(* CODESYS project TcTransform.library
   DefaultNamespace: TcTransform
   Description: Coordinate system transformation library
   Author: Andrew Burks
   DocFormat: reStructuredText
   Title: TcTransform
   Version: 0.3.36
   Company: Burks Engineering
   Placeholder: TcTransform

Project tree, tasks and I/O mapping:
  libraries: Tc2_Standard, * (Beckhoff Automation GmbH); Tc2_System, * (Beckhoff Automation GmbH); TcMatrix, 1.4.3 (Burks Engineering)
  DUTs/
    data type Dimension
    data type EulerAngleSequence
    data type TaitBryanAngleSequence
  POUs/
    AngleSequence/
      MatrixAccessors/
        function block AngleSequenceAccessor [ST]: Init, Cols, Rows
        function block AngleSequenceAngleAccessor [ST]: GetI, SetI
        function block AngleSequenceDimensionAccessor [ST]: GetI, SetI
      function block AngleSequenceOrientation [ST]: IsEqual, IsEqualDimension, IsEqualSize, IsNearlyEqual, GetAngle, GetDimension, GetRMatrix, AngleAccessor, DimensionAccessor, Length, Clear, SetAngle
      function block EulerAngleOrientation [ST]: GetAngle, GetDimension, GetDimensions, Length, RaDeg, RaRad, RbDeg, RbRad, RcDeg, RcRad, Sequence, Clear, CopyFrom, SetAngle, SetFromComponentsDeg, SetFromComponentsRad
      interface IAngleSequenceOrientation
      function block TaitBryanAngleOrientation [ST]: GetAngle, GetDimension, GetDimensions, Length, RxDeg, RxRad, RyDeg, RyRad, RzDeg, RzRad, Sequence, Clear, CopyFrom, SetAngle, SetFromComponentsDeg, SetFromComponentsRad, SetFromRMatrix
    Functions/
      function Vector3_CrossProduct [ST]
    function ATAN2 [ST]
    function block HMatrix [ST]: GetAngleSequenceComponent, GetReversed, GetTransformedHMatrix, GetTransformedHMatrixReverse, GetTransformedVector3, GetTransformedVector3Reverse, TransformHMatrix, TransformHMatrixReverse, TransformVector3, TransformVector3Reverse, OffsetBy, Reverse, RotateBy, RotateByReverse, TransformBy, TransformByReverse, Clear, FB_init, GetI, SetI, RMatrixAccessor, RMatrixComponent, Vector3Accessor, Vector3Component, SetFromComponents
    function block RMatrix [ST]: GetAngleSequence, GetReversed, GetRotatedRMatrix, GetRotatedRMatrixReverse, GetRotatedVector3, GetRotatedVector3Reverse, RotateRMatrix, RotateRMatrixReverse, RotateVector3, RotateVector3Reverse, Reverse, RotateBy, RotateByReverse, Clear, FB_init, GetI, SetI, ReversedAccessor, BuildFromUnitVectors, SetFromAngle, SetFromAngleSequence, SetFromVectorsXY, SetFromVectorsXZ, SetFromVectorsYZ
    function block Vector3 [ST]: GetReversed, GetVector3CrossProduct, GetVector3Difference, GetVector3DotProduct, GetVector3Scaled, GetVector3Sum, Reverse, RotateBy, RotateByReverse, SumWith, TransformBy, TransformByReverse, FB_init, GetI, SetI, X, Y, Z, SetAsCrossProduct, SetFromComponents
  Version/
    global variables Global_Version
*)

// DUTs/Dimension
{attribute 'qualified_only'}
{attribute 'strict'}
TYPE Dimension : 
(
	X := 0,
	Y := 1,
	Z := 2
)UINT;
END_TYPE

// DUTs/EulerAngleSequence
{attribute 'qualified_only'}
{attribute 'strict'}
TYPE EulerAngleSequence :
(
	ZXZ := 0,
	XYX := 1,
	YZY := 2,
	ZYZ := 3,
	XZX := 4,
	YXY := 5
);
END_TYPE

// DUTs/TaitBryanAngleSequence
{attribute 'qualified_only'}
{attribute 'strict'}
TYPE TaitBryanAngleSequence :
(
	XYZ := 0,
	YZX := 1,
	ZXY := 2,
	XZY := 3,
	ZYX := 4,
	YXZ := 5	//Standard Roll/Pitch/Yaw
);
END_TYPE

// Version/Global_Version
{attribute 'TcGenerated'}
{attribute 'no-analysis'}
{attribute 'linkalways'}
// This function has been automatically generated from the project information.
VAR_GLOBAL CONSTANT
	{attribute 'const_non_replaced'}
	stLibVersion_TcTransform : ST_LibVersion := (iMajor := 0, iMinor := 3, iBuild := 36, iRevision := 0, nFlags := 0, sVersion := '0.3.36');
END_VAR

// POUs/AngleSequence/MatrixAccessors/AngleSequenceAccessor
FUNCTION_BLOCK ABSTRACT AngleSequenceAccessor EXTENDS Matrix
VAR_INPUT
END_VAR
VAR_OUTPUT
END_VAR
VAR
	O_ : REFERENCE TO AngleSequenceOrientation;
END_VAR

METHOD PUBLIC Init
VAR_INPUT
	O : REFERENCE TO AngleSequenceOrientation;
END_VAR
O_ REF= O;
END_METHOD

//Total number of columns in this matrix
PROPERTY PUBLIC Cols : UINT
GET
IF NOT __ISVALIDREF(O_) THEN
	Cols := 0;
	LogWarning('%s Attempted Cols access using uninitialized Matrix Accessor');
ELSE
	Cols :=1;
END_IF
END_GET
END_PROPERTY

//Total number of rows in this matrix
PROPERTY PUBLIC Rows : UINT
GET
IF NOT __ISVALIDREF(O_) THEN
	Rows := 0;
	LogWarning('%s Attempted Rows access using uninitialized Matrix Accessor');
ELSE
	Rows := O_.Length;
END_IF;
END_GET
END_PROPERTY

END_FUNCTION_BLOCK

// POUs/AngleSequence/AngleSequenceOrientation
FUNCTION_BLOCK ABSTRACT AngleSequenceOrientation
VAR_INPUT
END_VAR
VAR_OUTPUT
END_VAR
VAR
	AngleAccessor_ : AngleSequenceAngleAccessor;
	DimensionAccessor_ : AngleSequenceDimensionAccessor;
END_VAR

METHOD PUBLIC IsEqual : BOOL
VAR_INPUT
	O : REFERENCE TO AngleSequenceOrientation;
END_VAR
IsEqual := IsEqualDimension(O) AND AngleAccessor.IsEqual(O.AngleAccessor);
END_METHOD

METHOD PUBLIC IsEqualDimension : BOOL
VAR_INPUT
	O : REFERENCE TO AngleSequenceOrientation;
END_VAR
IsEqualDimension := IsEqualSize(O) AND DimensionAccessor.IsEqual(O.DimensionAccessor);
END_METHOD

METHOD PUBLIC IsEqualSize : BOOL
VAR_INPUT
	O : REFERENCE TO AngleSequenceOrientation;
END_VAR
IsEqualSize := Length = O.Length;
END_METHOD

METHOD PUBLIC IsNearlyEqual : BOOL
VAR_INPUT
	O : REFERENCE TO AngleSequenceOrientation;
	Precision : LREAL;
END_VAR
IsNearlyEqual := IsEqualDimension(O) AND AngleAccessor.IsNearlyEqual(O.AngleAccessor, Precision);
END_METHOD

METHOD PUBLIC ABSTRACT GetAngle : LREAL
VAR_INPUT
	I : UINT;
END_VAR
END_METHOD

METHOD PUBLIC ABSTRACT GetDimension : Dimension
VAR_INPUT
	I : UINT;
END_VAR
END_METHOD

METHOD PUBLIC GetRMatrix : RMatrix
VAR_INPUT
END_VAR
VAR
	I : UINT;
	RTemp : RMatrix;
END_VAR
IF Length = 0 THEN
	RETURN;//identity
END_IF

//intrinsic rotations are chained left to right [https://en.wikipedia.org/wiki/Davenport_chained_rotations#Intrinsic_rotations]
//GetR := R_0 * R_1 * .. * R_n-1
//The best in-place function available is A := B * A (premultiplication) so we need to chain from n-1 to 0. Note that GetRMatrix is initialized to the identity
FOR I := 0 TO LENGTH-1 DO
	RTemp.SetFromAngle(GetAngle(Length-1-I),GetDimension(Length-1-I));
	GetRMatrix.RotateBy(RTemp);//premultiplication is intrinsic rotations
END_FOR
END_METHOD

//DO NOT HANG ON TO THIS POINTER. if you do assignment it won't carry over!
PROPERTY PUBLIC AngleAccessor : REFERENCE TO MATRIX
GET
AngleAccessor_.Init(THIS^);
AngleAccessor REF= AngleAccessor_;
END_GET
END_PROPERTY

//DO NOT HANG ON TO THIS POINTER. if you do assignment it won't carry over!
PROPERTY PUBLIC DimensionAccessor : REFERENCE TO MATRIX
GET
DimensionAccessor_.Init(THIS^);
DimensionAccessor REF= DimensionAccessor_;
END_GET
END_PROPERTY

PROPERTY PUBLIC ABSTRACT Length : UINT
GET
END_GET
END_PROPERTY

METHOD PUBLIC ABSTRACT Clear
VAR_INPUT
END_VAR
END_METHOD

METHOD PUBLIC ABSTRACT SetAngle : BOOL
VAR_INPUT
	I : UINT;
	Val : LREAL;
END_VAR
END_METHOD

END_FUNCTION_BLOCK

// POUs/AngleSequence/MatrixAccessors/AngleSequenceAngleAccessor
FUNCTION_BLOCK AngleSequenceAngleAccessor EXTENDS AngleSequenceAccessor
VAR_INPUT
END_VAR
VAR_OUTPUT
END_VAR
VAR
END_VAR

//Gets the value of the element in this matrix at the supplied location as if the elements were stored in a 1D row-major array
//:Prerequisites:
// - I < Rows*Cols
// - Matrix is not empty
//If the supplied index is out of bounds the value 0 is returned and a warning is generated in the Error List
METHOD PUBLIC GetI : LREAL//The value of the element at the specified index, or 0 if an invalid index is supplied
VAR_INPUT
	I : UINT;//The index of the element which should have its value returned
END_VAR
VAR
END_VAR
IF NOT __ISVALIDREF(O_) THEN
	GetI := 0.0;
	LogWarning('%s Attempted I access to uninitialized Matrix Accessor');
ELSIF IsEmpty THEN
	GetI := 0.0;
	LogWarning('%s: Attempted I access of empty Matrix Accessor');
ELSIF I >= Length THEN
	GetI := 0.0;
	LogWarning('%s: Attempted I access beyond limits of Matrix Accessor');
ELSE
	GetI := O_.GetAngle(I);
END_IF
END_METHOD

//Sets the element specified by the supplied index to the suppleid value, assuming the data of the matrix is stored in a 1D row-major array
//:Prerequisites: - I < Rows*Cols
METHOD PUBLIC SetI : BOOL//TRUE if the specified index is valid and the data is copied. FLASE otherwise
VAR_INPUT
	I : UINT;//The index specifying which element should be modified
	Val : LREAL;//The value copied to the corresponding element
END_VAR
IF NOT __ISVALIDREF(O_) THEN
	SetI := FALSE;
	LogWarning('%s Attempted I access to uninitialized Matrix Accessor');
ELSIF IsEmpty THEN
	SetI := FALSE;
	LogWarning('%s: Attempted I access of empty Matrix Accessor');
ELSIF I >= Length THEN
	SetI := FALSE;
	LogWarning('%s: Attempted I access beyond limits of Matrix Accessor');
ELSE
	SetI := TRUE;
	SetI := O_.SetAngle(I,Val);
END_IF
END_METHOD

END_FUNCTION_BLOCK

// POUs/AngleSequence/MatrixAccessors/AngleSequenceDimensionAccessor
FUNCTION_BLOCK AngleSequenceDimensionAccessor EXTENDS AngleSequenceAccessor
VAR_INPUT
END_VAR
VAR_OUTPUT
END_VAR
VAR
END_VAR

//Gets the value of the element in this matrix at the supplied location as if the elements were stored in a 1D row-major array
//:Prerequisites:
// - I < Rows*Cols
// - Matrix is not empty
//If the supplied index is out of bounds the value 0 is returned and a warning is generated in the Error List
METHOD PUBLIC GetI : LREAL//The value of the element at the specified index, or 0 if an invalid index is supplied
VAR_INPUT
	I : UINT;//The index of the element which should have its value returned
END_VAR
VAR
END_VAR
IF NOT __ISVALIDREF(O_) THEN
	GetI := 0.0;
	LogWarning('%s Attempted I access to uninitialized Matrix Accessor');
ELSIF IsEmpty THEN
	GetI := 0.0;
	LogWarning('%s: Attempted I access of empty Matrix Accessor');
ELSIF I >= Length THEN
	GetI := 0.0;
	LogWarning('%s: Attempted I access beyond limits of Matrix Accessor');
ELSE
	GetI := UINT_TO_LREAL(O_.GetDimension(I));
END_IF
END_METHOD

//Sets the element specified by the supplied index to the suppleid value, assuming the data of the matrix is stored in a 1D row-major array
//:Prerequisites: - I < Rows*Cols
METHOD PUBLIC SetI : BOOL//TRUE if the specified index is valid and the data is copied. FLASE otherwise
VAR_INPUT
	I : UINT;//The index specifying which element should be modified
	Val : LREAL;//The value copied to the corresponding element
END_VAR
SetI := FALSE;//READ ONLY!!!
END_METHOD

END_FUNCTION_BLOCK

// POUs/RMatrix
(*
RMatrix : 3D Rotation Matrix
======================

Overview
----------------------

This class represents a 3x3 matrix used to represent a rotation.

See: `https://en.wikipedia.org/wiki/Rotation_matrix`__

You can think of the RMatrix as representing the orientation of  *child* coordinate system inside a *parent* coordinate system. 
Each column vector of the RMatrix is essentially a unit vector (X, Y, or Z) of the child coordinate system projected into the parent coordinate system.
Premultiplication with this matrix transforms vectors and other rotations out of the child coordinate system and into the parent coordinate system. 
Reversing the RMatrix simply reverses the roles (parent/child) of the coordinate system and allows transformations in the other direction.
*)
{attribute 'reflection'}
FUNCTION_BLOCK RMatrix EXTENDS StaticMatrix
VAR_INPUT
END_VAR
VAR_OUTPUT
END_VAR
VAR
	Data : ARRAY[0..cRows*cCols-1] OF LREAL;
	ReversedAccessor_ : TransposeMatrixAccessor;//reinitialize every use (via property) because := copying will destroy the pointer
END_VAR
VAR CONSTANT
	cRows : UINT := 3;
	cCols : UINT := 3;
END_VAR

//Returns a ZYX tait-Bryan angle sequence that represents this rotation matrix
METHOD PUBLIC GetAngleSequence : TaitBryanAngleOrientation
VAR_INPUT
END_VAR
GetAngleSequence.SetFromRMatrix(THIS^);
END_METHOD

METHOD PUBLIC GetReversed : RMatrix
VAR_INPUT
END_VAR
GetReversed := THIS^;
GetReversed.Reverse();
END_METHOD

METHOD PUBLIC GetRotatedRMatrix : RMatrix;
VAR_INPUT
	M_R : RMatrix;
END_VAR
RotateRMatrix(M_R,GetRotatedRMatrix);
END_METHOD

METHOD PUBLIC GetRotatedRMatrixReverse : RMatrix;
VAR_INPUT
	M_R : RMatrix;
END_VAR
RotateRMatrixReverse(M_R,GetRotatedRMatrixReverse);
END_METHOD

METHOD PUBLIC GetRotatedVector3 : Vector3
VAR_INPUT
	M_V : Vector3;
END_VAR
RotateVector3(M_V,GetRotatedVector3);
END_METHOD

METHOD PUBLIC GetRotatedVector3Reverse : Vector3
VAR_INPUT
	M_V : Vector3;
END_VAR
RotateVector3Reverse(M_V,GetRotatedVector3Reverse);
END_METHOD

METHOD PUBLIC RotateRMatrix
VAR_INPUT
	R_From : RMatrix;
	R_To : REFERENCE TO RMatrix;
END_VAR
Matrix_Product(THIS^,R_From,R_To);
END_METHOD

METHOD PUBLIC RotateRMatrixReverse
VAR_INPUT
	R_From : RMatrix;
	R_To : REFERENCE TO RMatrix;
END_VAR
Matrix_Product(ReversedAccessor,R_From,R_To);
END_METHOD

METHOD PUBLIC RotateVector3
VAR_INPUT
	V_From : Vector3;
	V_To : REFERENCE TO Vector3;
END_VAR
Matrix_Product(THIS^,V_From,V_To);
END_METHOD

METHOD PUBLIC RotateVector3Reverse
VAR_INPUT
	V_From : Vector3;
	V_To : REFERENCE TO Vector3;
END_VAR
Matrix_Product(ReversedAccessor,V_From,V_To);
END_METHOD

METHOD PUBLIC Reverse
VAR_INPUT
END_VAR
Matrix_TransposeSquare(THIS^);
END_METHOD

//Equivalent to Matrix Operation 'THIS := M_R * THIS'
METHOD PUBLIC RotateBy
VAR_INPUT
	M_R : RMatrix;
END_VAR
VAR
	Temp : RMatrix := THIS^;
END_VAR
M_R.RotateRMatrix(Temp,THIS^);
END_METHOD

//Equivalent to Matrix Operation 'THIS := M_R * THIS'
METHOD PUBLIC RotateByReverse
VAR_INPUT
	M_R : RMatrix;
END_VAR
VAR
	Temp : RMatrix := THIS^;
END_VAR
M_R.RotateRMatrixReverse(Temp,THIS^);
END_METHOD

METHOD PUBLIC Clear
VAR_INPUT
END_VAR
FillTrapezoidal(1,0,0);
END_METHOD

METHOD FB_init : BOOL
VAR_INPUT
	bInitRetains : BOOL; // if TRUE, the retain variables are initialized (warm start / cold start)
	bInCopyCode : BOOL;  // if TRUE, the instance afterwards gets moved into the copy code (online change)
END_VAR
Init_(cRows,cCols);
Clear();
END_METHOD

//Gets the value of the element in this matrix at the supplied location as if the elements were stored in a 1D row-major array
//:Prerequisites:
// - I < Rows*Cols
// - Matrix is not empty
//If the supplied index is out of bounds the value 0 is returned and a warning is generated in the Error List
METHOD PUBLIC GetI : LREAL//The value of the element at the specified index, or 0 if an invalid index is supplied
VAR_INPUT
	I : UINT;//The index of the element which should have its value returned
END_VAR
IF I >= Length THEN
	GetI := 0.0;
	LogWarning('%s: Attempted I access of out-of-bounds Matrix data');
ELSE
	GetI := Data[I];
END_IF
END_METHOD

//Sets the element specified by the supplied index to the suppleid value, assuming the data of the matrix is stored in a 1D row-major array
//:Prerequisites: - I < Rows*Cols
METHOD PUBLIC SetI : BOOL//TRUE if the specified index is valid and the data is copied. FLASE otherwise
VAR_INPUT
	I : UINT;//The index specifying which element should be modified
	Val : LREAL;//The value copied to the corresponding element
END_VAR
IF I >= Length THEN
	SetI := FALSE;
	LogWarning('%s: Attempt to set data using I access when I is out of bounds');
ELSE
	SetI := TRUE;
	Data[I] := Val;
END_IF
END_METHOD

PROPERTY PROTECTED ReversedAccessor : REFERENCE TO Matrix
GET
ReversedAccessor_.Init(THIS^);
ReversedAccessor REF= ReversedAccessor_;
END_GET
END_PROPERTY

METHOD PROTECTED BuildFromUnitVectors
VAR_INPUT
	X : Vector3;
	Y : Vector3;
	Z : Vector3;
END_VAR
FillFromAt(X,0,0);
FillFromAt(Y,0,1);
FillFromAt(Z,0,2);
END_METHOD

METHOD PUBLIC SetFromAngle
VAR_INPUT
	Angle : LREAL;//radians
	Dimension : Dimension;//0-2
END_VAR
VAR
	SM : ShrunkMatrixAccessor;
	Sign : LREAL;
	
END_VAR
FillTrapezoidal(1,0,0);
Sign := INT_TO_LREAL(((UINT_TO_INT(Dimension) MOD 2)*2)-1);
SM := GetShrunkMatrixAccessor(Dimension,Dimension);
SM.FillTrapezoidal(COS(Angle),Sign*SIN(Angle),-1*Sign*SIN(Angle));
END_METHOD

//Intrinsic Rotations
METHOD PUBLIC SetFromAngleSequence
VAR_INPUT
END_VAR
VAR_IN_OUT
	Angles : ARRAY [*] OF LREAL;
	Dimensions : ARRAY [*] OF Dimension;
END_VAR
VAR
	I : DINT;
	N : DINT;
	RTemp : RMatrix;
END_VAR
N := MIN(UPPER_BOUND(Angles,1) - LOWER_BOUND(Angles,1),UPPER_BOUND(Dimensions,1) - LOWER_BOUND(Dimensions,1))+1;
FillTrapezoidal(1,0,0);
FOR I := N-1 TO 0 BY -1 DO
	RTemp.SetFromAngle(Angles[LOWER_BOUND(Angles,1)+I],Dimensions[LOWER_BOUND(Dimensions,1)+I]);
	RotateBy(RTemp);
END_FOR
END_METHOD

METHOD PUBLIC SetFromVectorsXY
VAR_INPUT
	X : VEctor3;//make a copy so we can nromalize
	Y : Vector3;//make a copy so we can normalize
END_VAR
VAR
	Z : Vector3;
END_VAR
X.Normalize();
Y.Normalize();
IF ABS(X.GetVector3DotProduct(Y)) > 1E-9 THEN
	LogWarning('%s: the two vectors used to construct the coordinate system were not perpendicular');
END_IF
Z.SetAsCrossProduct(X,Y);
BuildFromUnitVectors(X,Y,Z);
END_METHOD

METHOD PUBLIC SetFromVectorsXZ
VAR_INPUT
	X : VEctor3;//make a copy so we can nromalize
	Z : Vector3;//make a copy so we can normalize
END_VAR
VAR
	Y : Vector3;
END_VAR
X.Normalize();
Z.Normalize();
IF ABS(X.GetVector3DotProduct(Y)) > 1E-9 THEN
	LogWarning('%s: the two vectors used to construct the coordinate system were not perpendicular');
END_IF
Y.SetAsCrossProduct(Z,X);
BuildFromUnitVectors(X,Y,Z);
END_METHOD

METHOD PUBLIC SetFromVectorsYZ
VAR_INPUT
	Y : VEctor3;//make a copy so we can nromalize
	Z : Vector3;//make a copy so we can normalize
END_VAR
VAR
	X : Vector3;
END_VAR
Y.Normalize();
Z.Normalize();
IF ABS(X.GetVector3DotProduct(Y)) > 1E-9 THEN
	LogWarning('%s: the two vectors used to construct the coordinate system were not perpendicular');
END_IF
X.SetAsCrossProduct(Y,Z);
BuildFromUnitVectors(X,Y,Z);
END_METHOD

END_FUNCTION_BLOCK

// POUs/AngleSequence/TaitBryanAngleOrientation
FUNCTION_BLOCK TaitBryanAngleOrientation EXTENDS AngleSequenceOrientation
VAR_INPUT
END_VAR
VAR_OUTPUT
END_VAR
VAR
	Angles_ : ARRAY [0..2] OF LREAL;
	Sequence_ : TaitBryanAngleSequence;
END_VAR

METHOD PUBLIC  GetAngle : LREAL
VAR_INPUT
	I : UINT;
END_VAR
VAR
	Dim : Dimension;
END_VAR
IF I >= Length THEN
	GetAngle := 0;
	RETURN;
END_IF

Dim := GetDimension(I);

IF Dim >= Length THEN
	GetAngle := 0;
	RETURN;
END_IF

GetAngle := Angles_[Dim];
END_METHOD

METHOD PUBLIC GetDimension : Dimension
VAR_INPUT
	I : UINT;
END_VAR
VAR
	Dims : ARRAY [0..2] OF Dimension;
END_VAR
IF I >= Length THEN
	GetDimension := 0;
	RETURN;
END_IF

Dims := GetDimensions();
GetDimension := Dims[I];
END_METHOD

METHOD PUBLIC GetDimensions : ARRAY [0..2] OF Dimension
VAR_INPUT
END_VAR
CASE Sequence OF
	TaitBryanAngleSequence.XYZ:
		GetDimensions[0] := 0;
		GetDimensions[1] := 1;
		GetDimensions[2] := 2;
	TaitBryanAngleSequence.XZY:
		GetDimensions[0] := 0;
		GetDimensions[1] := 2;
		GetDimensions[2] := 1;
	TaitBryanAngleSequence.YXZ:
		GetDimensions[0] := 1;
		GetDimensions[1] := 0;
		GetDimensions[2] := 2;
	TaitBryanAngleSequence.YZX:
		GetDimensions[0] := 1;
		GetDimensions[1] := 2;
		GetDimensions[2] := 0;
	TaitBryanAngleSequence.ZXY:
		GetDimensions[0] := 2;
		GetDimensions[1] := 0;
		GetDimensions[2] := 1;
	TaitBryanAngleSequence.ZYX:
		GetDimensions[0] := 2;
		GetDimensions[1] := 1;
		GetDimensions[2] := 0;
	ELSE
		GetDimensions[0] := 0;
		GetDimensions[1] := 0;
		GetDimensions[2] := 0;
END_CASE
END_METHOD

PROPERTY Length : UINT
GET
Length := 3;
END_GET
END_PROPERTY

PROPERTY PUBLIC RxDeg : LREAL
GET
RxDeg := 180 * Angles_[0] / PI;
END_GET
SET
Angles_[0] := PI * RxDeg / 180;
END_SET
END_PROPERTY

PROPERTY PUBLIC RxRad : LREAL
GET
RxRad := Angles_[0];
END_GET
SET
Angles_[0] := RxRad;
END_SET
END_PROPERTY

PROPERTY PUBLIC RyDeg : LREAL
GET
RyDeg := 180 * Angles_[1] / PI;
END_GET
SET
Angles_[1] := PI * RyDeg / 180;
END_SET
END_PROPERTY

PROPERTY PUBLIC RyRad : LREAL
GET
RyRad := Angles_[1];
END_GET
SET
Angles_[1] := RyRad;
END_SET
END_PROPERTY

PROPERTY PUBLIC RzDeg : LREAL
GET
RzDeg := 180 * Angles_[2] / PI;
END_GET
SET
Angles_[2] := PI * RzDeg / 180;
END_SET
END_PROPERTY

PROPERTY PUBLIC RzRad : LREAL
GET
RzRad := Angles_[2];
END_GET
SET
Angles_[2] := RzRad;
END_SET
END_PROPERTY

PROPERTY PUBLIC Sequence : TaitBryanAngleSequence
GET
Sequence := Sequence_;
END_GET
SET
Sequence_ := Sequence;
END_SET
END_PROPERTY

METHOD PUBLIC Clear
VAR_INPUT
END_VAR
Angles_[0] := 0;
Angles_[1] := 0;
Angles_[2] := 0;
END_METHOD

METHOD PUBLIC CopyFrom
VAR_INPUT
	O : TaitBryanAngleOrientation;
END_VAR
Clear();
Sequence := O.Sequence;
AngleAccessor.CopyFrom(O.AngleAccessor);
END_METHOD

METHOD PUBLIC SetAngle : BOOL
VAR_INPUT
	I : UINT;
	Val : LREAL;
END_VAR
VAR
	Dim : Dimension;
END_VAR
IF I >= Length THEN
	SetAngle := FALSE;
	RETURN;
END_IF

Dim := GetDimension(I);

IF Dim >= Length THEN
	SetAngle := FALSE;
	RETURN;
END_IF

SetAngle := TRUE;

Angles_[Dim] := Val;
END_METHOD

METHOD PUBLIC SetFromComponentsDeg
VAR_INPUT
	Rx : LREAL;
	Ry : LREAL;
	Rz : LREAL;
	Seq : TaitBryanAngleSequence;
END_VAR
RxDeg := Rx;
RyDeg := Ry;
RzDeg := Rz;
Sequence := Seq;
END_METHOD

METHOD PUBLIC SetFromComponentsRad
VAR_INPUT
	Rx : LREAL;
	Ry : LREAL;
	Rz : LREAL;
	Seq : TaitBryanAngleSequence;
END_VAR
RxRad := Rx;
RyRad := Ry;
RzRad := Rz;
Sequence := Seq;
END_METHOD

METHOD PUBLIC SetFromRMatrix
VAR_INPUT
	M_R : RMatrix;
END_VAR
Sequence := TaitBryanAngleSequence.ZYX;
IF M_R.GetRC(0,0) = 0 AND M_R.GetRC(1,0) = 0 THEN
	RzRad := 0;
	RyRad := PI/2;
	RxRad := ATAN2(M_R.GetRC(0,1),M_R.GetRC(1,1));
ELSE
	RzRad := ATAN2(M_R.GetRC(1,0),M_R.GETRC(0,0));
	RyRad := ATAN2(-1*M_R.GetRC(2,0),SQRT(M_R.GetRC(0,0)*M_R.GetRC(0,0) + M_R.GetRC(1,0)*M_R.GetRC(1,0)));
	RxRad := ATAN2(M_R.GetRC(2,1),M_R.GetRC(2,2));
END_IF
END_METHOD

END_FUNCTION_BLOCK

// POUs/ATAN2
//ATAN2(Y,X); [https://en.wikipedia.org/wiki/Atan2]
FUNCTION ATAN2 : LREAL
VAR_INPUT
	Y : LREAL;
	X : LREAL;
END_VAR
VAR
END_VAR

IF X > 0 THEN
	ATAN2 := ATAN(Y/X);
ELSIF X < 0 AND Y >= 0 THEN
	ATAN2 := ATAN(Y/X) + PI;
ELSIF X < 0 AND Y < 0 THEN
	ATAN2 := ATAN(Y/X) - PI;
ELSIF X = 0 AND Y > 0 THEN
	ATAN2 := PI/2;
ELSIF X = 0 AND Y < 0 THEN
	ATAN2 := -PI/2;
ELSE //X=0 AND y=0
	//technically undefined...
	ATAN2 := 0;
	ADSLOGSTR(ADSLOG_MSGTYPE_WARN,'Attempt to use ATAN2 with X=0 and Y=0 detected. Function is undefined for this case!','');
END_IF

END_FUNCTION

// POUs/Vector3
(*
Vector3 : 3D Position Vector
======================

Overview
----------------------

This class represents a 3x1 column vector used to represent the position of a point within a coordinate system.

*)
{attribute 'reflection'}
FUNCTION_BLOCK Vector3 EXTENDS StaticMatrix
VAR_INPUT
END_VAR
VAR_OUTPUT
END_VAR
VAR
	Data : ARRAY[0..cRows*cCols-1] OF LREAL;
END_VAR
VAR CONSTANT
	cRows : UINT := 3;
	cCols : UINT := 1;
END_VAR

METHOD PUBLIC GetReversed : Vector3
VAR_INPUT
END_VAR
GetReversed := THIS^;
GetReversed.Reverse();
END_METHOD

//Equivalent to Result := THIS x M_V
METHOD PUBLIC GetVector3CrossProduct : Vector3
VAR_INPUT
	M_V : Vector3;
END_VAR
Vector3_CrossProduct(This^,M_V,GetVector3CrossProduct);
END_METHOD

METHOD PUBLIC GetVector3Difference : Vector3
VAR_INPUT
	M_V : Vector3;
END_VAR
Matrix_ElementDifference(THIS^,M_V,GetVector3Difference);
END_METHOD

METHOD PUBLIC GetVector3DotProduct : LREAL
VAR_INPUT
	M_V : Vector3;
END_VAR
GetVector3DotProduct := GetVectorDotProduct(M_V);
END_METHOD

METHOD PUBLIC GetVector3Scaled : Vector3
VAR_INPUT
	Scalar : LREAL;
END_VAR
GetVector3Scaled := THIS^;
GetVector3Scaled.Scale(Scalar);
END_METHOD

METHOD PUBLIC GetVector3Sum : Vector3
VAR_INPUT
	M_V : Vector3;
END_VAR
Matrix_ElementSum(THIS^,M_V,GetVector3Sum);
END_METHOD

METHOD PUBLIC Reverse
VAR_INPUT
END_VAR
Scale(-1);
END_METHOD

METHOD PUBLIC RotateBy
VAR_INPUT
	M_R : RMAtrix;
END_VAR
VAR
	Temp : Vector3 := THIS^;
END_VAR
M_R.RotateVector3(Temp,THIS^);
END_METHOD

METHOD PUBLIC RotateByReverse
VAR_INPUT
	M_R : RMAtrix;
END_VAR
VAR
	Temp : Vector3 := THIS^;
END_VAR
M_R.RotateVector3Reverse(Temp,THIS^);
END_METHOD

METHOD PUBLIC SumWith
VAR_INPUT
	M_V : Vector3;
END_VAR
Matrix_ElementSum(THIS^,M_V,THIS^);
END_METHOD

METHOD PUBLIC TransformBy
VAR_INPUT
	M_H : HMatrix;
END_VAR
VAR
	Temp : Vector3 := THIS^;
END_VAR
M_H.TransformVector3(temp,THIS^);
END_METHOD

METHOD PUBLIC TransformByReverse
VAR_INPUT
	M_H : HMatrix;
END_VAR
VAR
	Temp : Vector3 := THIS^;
END_VAR
M_H.TransformVector3Reverse(Temp,THIS^);
END_METHOD

METHOD FB_init : BOOL
VAR_INPUT
	bInitRetains : BOOL; // if TRUE, the retain variables are initialized (warm start / cold start)
	bInCopyCode : BOOL;  // if TRUE, the instance afterwards gets moved into the copy code (online change)
END_VAR
Init_(cRows,cCols);
Clear();
END_METHOD

//Gets the value of the element in this matrix at the supplied location as if the elements were stored in a 1D row-major array
//:Prerequisites:
// - I < Rows*Cols
// - Matrix is not empty
//If the supplied index is out of bounds the value 0 is returned and a warning is generated in the Error List
METHOD PUBLIC GetI : LREAL//The value of the element at the specified index, or 0 if an invalid index is supplied
VAR_INPUT
	I : UINT;//The index of the element which should have its value returned
END_VAR
IF I >= Length THEN
	GetI := 0.0;
	LogWarning('%s: Attempted I access of out-of-bounds Matrix data');
ELSE
	GetI := Data[I];
END_IF
END_METHOD

//Sets the element specified by the supplied index to the suppleid value, assuming the data of the matrix is stored in a 1D row-major array
//:Prerequisites: - I < Rows*Cols
METHOD PUBLIC SetI : BOOL//TRUE if the specified index is valid and the data is copied. FLASE otherwise
VAR_INPUT
	I : UINT;//The index specifying which element should be modified
	Val : LREAL;//The value copied to the corresponding element
END_VAR
IF I >= Length THEN
	SetI := FALSE;
	LogWarning('%s: Attempt to set data using I access when I is out of bounds');
ELSE
	SetI := TRUE;
	Data[I] := Val;
END_IF
END_METHOD

PROPERTY PUBLIC X : LREAL
GET
X := GetI(0);
END_GET
SET
SetI(0,X);
END_SET
END_PROPERTY

PROPERTY PUBLIC Y : LREAL
GET
Y := GetI(1);
END_GET
SET
SetI(1,Y);
END_SET
END_PROPERTY

PROPERTY PUBLIC Z : LREAL
GET
Z := GetI(2);
END_GET
SET
SetI(2,Z);
END_SET
END_PROPERTY

METHOD PUBLIC SetAsCrossProduct
VAR_INPUT
	A : Vector3;
	B : Vector3;
END_VAR
VAR
	Vs : ARRAY[0..1] OF POINTER TO MATRIX;
END_VAR
Vector3_CrossProduct(A,B,This^);
END_METHOD

METHOD PUBLIC SetFromComponents
VAR_INPUT
	Xp : LREAL;
	Yp : LREAL;
	Zp : LREAL;
END_VAR
X := Xp;
Y := Yp;
Z := Zp;
END_METHOD

END_FUNCTION_BLOCK

// POUs/Functions/Vector3_CrossProduct
//Specialized, optimized version of the generic vector cross product specifically for vector 3
//Thanks to captain-yoshi for the algorithm and idea
//see https://github.com/BurksEngineering/TcTransform/issues/4
FUNCTION Vector3_CrossProduct
VAR_IN_OUT CONSTANT
    A : Vector3;
    B : Vector3;
END_VAR
VAR_IN_OUT
    Res : Vector3;
END_VAR

// Complexity : 6M+3A
Res.SetI(0, A.GetI(1)*B.GetI(2) - A.GetI(2)*B.GetI(1));
Res.SetI(1, A.GetI(2)*B.GetI(0) - A.GetI(0)*B.GetI(2));
Res.SetI(2, A.GetI(0)*B.GetI(1) - A.GetI(1)*B.GetI(0));

END_FUNCTION

// POUs/HMatrix
(*
HMatrix : 3D Homogeneous Transformation Matrix
======================

Overview
----------------------

This class represents a 4x4 matrix used to represent the relative position and orientation of two coordinate system.

See: `http://planning.cs.uiuc.edu/node111.html`__

You can think of the HMatrix as representing the position and orientation of  *child* coordinate system inside a *parent* coordinate system.\
The included 3x3 matrix in the top left of the HMatrix is simply an RMatrix describing the relative angle, while the included 3x1 column vector in the top right of the HMatrix is simply a Vector3 describing the relative position.
Premultiplication with this matrix transforms vectors and coordiante systems out of the child coordinate system and into the parent coordinate system. 
Reversing the HMatrix simply reverses the roles (parent/child) of the coordinate system and allows transformations in the other direction.
*)
{attribute 'reflection'}
FUNCTION_BLOCK HMatrix EXTENDS StaticMatrix
VAR_INPUT
END_VAR
VAR_OUTPUT
END_VAR
VAR
	Data : ARRAY[0..cRows*cCols-1] OF LREAL;
	RMatrixAccessor_ : SubMatrixAccessor;//reinitialize every use (via property) because := copying will destroy the pointer
	Vector3Accessor_ : SubMatrixAccessor;//reinitialize every use (via property) because := copying will destroy the pointer
END_VAR
VAR CONSTANT
	cRows : UINT := 4;
	cCols : UINT := 4;
END_VAR

METHOD PUBLIC GetAngleSequenceComponent : TaitBryanAngleOrientation
VAR_INPUT
END_VAR
GetAngleSequenceComponent.SetFromRMatrix(RMatrixComponent);
END_METHOD

METHOD PUBLIC GetReversed : HMatrix
VAR_INPUT
END_VAR
GetReversed.CopyFrom(THIS^);
GetReversed.Reverse();
END_METHOD

//Equivalent to matrix multiplication: RETVAL = THIS * M_H
//CinA := BinA.GetTransformedHMatrix(CinB)
//CinA := BinA.GetTransformedHMatrix(BinC.GetReversed())
METHOD PUBLIC GetTransformedHMatrix : HMatrix
VAR_INPUT
	M_H : HMatrix;
END_VAR
TransformHMatrix(M_H,GetTransformedHMatrix);
END_METHOD

//Equivalent to matrix multiplication: RETVAL = THIS' * M_H
//CinA := AinB.GetTransformedHMatrixReverse(CinB)
//CinA := AinB.GetTransformedHMatrixReverse(BinC.GetReversed())
METHOD PUBLIC GetTransformedHMatrixReverse : HMatrix
VAR_INPUT
	M_H : HMatrix;
END_VAR
VAR
END_VAR
TransformHMatrixReverse(M_H,GetTransformedHMatrixReverse);
END_METHOD

METHOD PUBLIC GetTransformedVector3 : Vector3
VAR_INPUT
	M_V : Vector3;
END_VAR
VAR
	V4_in : ExternalStaticMatrix;
	V4_Data_in : ARRAY[0..3] OF LREAL;
	
	V4_out : ExternalStaticMatrix;
	V4_Data_out : ARRAY[0..3] OF LREAL;
END_VAR
TransformVector3(M_V,GetTransformedVector3);
END_METHOD

METHOD PUBLIC GetTransformedVector3Reverse : Vector3
VAR_INPUT
	M_V : Vector3;
END_VAR
VAR
	V4_in : ExternalStaticMatrix;
	V4_Data_in : ARRAY[0..3] OF LREAL;
	
	V4_out : ExternalStaticMatrix;
	V4_Data_out : ARRAY[0..3] OF LREAL;
END_VAR
TransformVector3Reverse(M_V,GetTransformedVector3Reverse);
END_METHOD

//Equivalent to matrix multiplication: H_To = THIS * H_From
//BinA.TransformHMatrix(CinB, out => CinA)
//BinA.TransformHMatrix(BinC.GetReversed(), out => CinA)
METHOD PUBLIC TransformHMatrix
VAR_INPUT
	H_From : HMatrix;
	H_To : REFERENCE TO HMatrix;
END_VAR
Matrix_Product(THIS^,H_From,H_To);
END_METHOD

//Equivalent to matrix multiplication: H_To = THIS' * H_From
//AinB.TransformHMatrixReverse(CinB, out => CinA)
//AinB.TransformHMatrixReverse(BinC.GetReversed(), out => CinA)
METHOD PUBLIC TransformHMatrixReverse
VAR_INPUT
	H_From : HMatrix;
	H_To : REFERENCE TO HMatrix;
END_VAR
VAR
	Temp : HMatrix;
END_VAR
Temp := GetReversed();
Matrix_Product(TEmp,H_From,H_To);
END_METHOD

METHOD PUBLIC TransformVector3
VAR_INPUT
	V_From : Vector3;
	V_To : REFERENCE TO Vector3;
END_VAR
VAR
	V4_in : ExternalStaticMatrix;
	V4_Data_in : ARRAY[0..3] OF LREAL;
	
	V4_out : ExternalStaticMatrix;
	V4_Data_out : ARRAY[0..3] OF LREAL;
END_VAR
V4_in.Init(ADR(V4_Data_in),4,1);
V4_in.FillFrom(V_From);
V4_in.SetI(3,1);

V4_out.Init(ADR(V4_Data_out),4,1);

Matrix_Product(THIS^,V4_in,V4_out);

V_To.FillFrom(V4_out);
END_METHOD

METHOD PUBLIC TransformVector3Reverse
VAR_INPUT
	V_From : Vector3;
	V_To : REFERENCE TO Vector3;
END_VAR
VAR
	V4_in : ExternalStaticMatrix;
	V4_Data_in : ARRAY[0..3] OF LREAL;
	
	Temp : HMatrix;
	
	V4_out : ExternalStaticMatrix;
	V4_Data_out : ARRAY[0..3] OF LREAL;
END_VAR
V4_in.Init(ADR(V4_Data_in),4,1);
V4_in.FillFrom(V_From);
V4_in.SetI(3,1);

V4_out.Init(ADR(V4_Data_out),4,1);

Temp := GetReversed();
Matrix_Product(temp,V4_in,V4_out);

V_To.FillFrom(V4_out);
END_METHOD

METHOD PUBLIC OffsetBy
VAR_INPUT
	In : Vector3;
END_VAR
VAR
	
END_VAR
Matrix_ElementSum(In,Vector3Accessor,Vector3Accessor);
END_METHOD

METHOD PUBLIC Reverse
VAR_INPUT
END_VAR
VAR
	Vtemp : Vector3;
END_VAR
Matrix_TransposeSquare(RMatrixAccessor);
Vtemp := Vector3Component;
Matrix_Product(RMatrixAccessor,Vtemp,Vector3Accessor);
Matrix_Scale(Vector3Accessor,-1);
END_METHOD

METHOD PUBLIC RotateBy
VAR_INPUT
	In : RMatrix;
END_VAR
VAR
	NewR : RMatrix;
END_VAR
Matrix_Product(In,RMatrixAccessor,NewR);
RMatrixAccessor.CopyFrom(NewR);
END_METHOD

METHOD PUBLIC RotateByReverse
VAR_INPUT
	In : RMatrix;
END_VAR
VAR
	InRev : RMatrix;
	TempRes : RMatrix;
END_VAR
InRev := In.GetReversed();
Matrix_Product(InRev,RmatrixAccessor,TempRes);
RMatrixAccessor.CopyFrom(TempRes);
END_METHOD

//Equivalent to Matrix Operation 'THIS := M_H * THIS'
METHOD PUBLIC TransformBy
VAR_INPUT
	M_H : HMatrix;
END_VAR
VAR
	Temp : HMatrix := THIS^;
END_VAR
M_H.TransformHMatrix(Temp,THIS^);
END_METHOD

//Equivalent to Matrix Operation 'THIS := M_H * THIS'
METHOD PUBLIC TransformByReverse
VAR_INPUT
	M_H : HMatrix;
END_VAR
VAR
	Temp : HMatrix := THIS^;
END_VAR
M_H.TransformHMatrixReverse(Temp,THIS^);
END_METHOD

METHOD PUBLIC Clear
VAR_INPUT
END_VAR
FillTrapezoidal(1,0,0);
END_METHOD

METHOD FB_init : BOOL
VAR_INPUT
	bInitRetains : BOOL; // if TRUE, the retain variables are initialized (warm start / cold start)
	bInCopyCode : BOOL;  // if TRUE, the instance afterwards gets moved into the copy code (online change)
END_VAR
Init_(cRows,cCols);
Clear();
END_METHOD

//Gets the value of the element in this matrix at the supplied location as if the elements were stored in a 1D row-major array
//:Prerequisites:
// - I < Rows*Cols
// - Matrix is not empty
//If the supplied index is out of bounds the value 0 is returned and a warning is generated in the Error List
METHOD PUBLIC GetI : LREAL//The value of the element at the specified index, or 0 if an invalid index is supplied
VAR_INPUT
	I : UINT;//The index of the element which should have its value returned
END_VAR
IF I >= Length THEN
	GetI := 0.0;
	LogWarning('%s: Attempted I access of out-of-bounds Matrix data');
ELSE
	GetI := Data[I];
END_IF
END_METHOD

//Sets the element specified by the supplied index to the suppleid value, assuming the data of the matrix is stored in a 1D row-major array
//:Prerequisites: - I < Rows*Cols
METHOD PUBLIC SetI : BOOL//TRUE if the specified index is valid and the data is copied. FLASE otherwise
VAR_INPUT
	I : UINT;//The index specifying which element should be modified
	Val : LREAL;//The value copied to the corresponding element
END_VAR
IF I >= Length THEN
	SetI := FALSE;
	LogWarning('%s: Attempt to set data using I access when I is out of bounds');
ELSE
	SetI := TRUE;
	Data[I] := Val;
END_IF
END_METHOD

//destroy immediately after use because if you ever := copy this FB the pointer within the accessor will still point to the old copy!!!!
PROPERTY PROTECTED RMatrixAccessor : REFERENCE TO SubMatrixAccessor
GET
RMatrixAccessor_.Init(THIS^,0,3,0,3);
RMatrixAccessor REF= RMatrixAccessor_;
END_GET
END_PROPERTY

PROPERTY PUBLIC RMatrixComponent : RMatrix
GET
RMatrixComponent.CopyFrom(RMatrixAccessor);
END_GET
SET
RMatrixAccessor.CopyFrom(RMatrixComponent);
END_SET
END_PROPERTY

//destroy immediately after use because if you ever := copy this FB the pointer within the accessor will still point to the old copy!!!!
PROPERTY PROTECTED Vector3Accessor : REFERENCE TO SubMatrixAccessor
GET
Vector3Accessor_.Init(THIS^,0,3,3,1);
Vector3Accessor REF= Vector3Accessor_;
END_GET
END_PROPERTY

PROPERTY PUBLIC Vector3Component : Vector3
GET
Vector3Component.CopyFrom(Vector3Accessor);
END_GET
SET
Vector3Accessor.CopyFrom(Vector3Component);
END_SET
END_PROPERTY

METHOD PUBLIC SetFromComponents
VAR_INPUT
	M_R : RMatrix;
	M_V : Vector3;
END_VAR
Clear();
M_R.CopyTo(RMatrixAccessor);
M_V.CopyTo(Vector3Accessor);
END_METHOD

END_FUNCTION_BLOCK

// POUs/AngleSequence/EulerAngleOrientation
FUNCTION_BLOCK EulerAngleOrientation EXTENDS AngleSequenceOrientation
VAR_INPUT
END_VAR
VAR_OUTPUT
END_VAR
VAR
	Angles_ : ARRAY [0..2] OF LREAL; 
	Sequence_ : EulerAngleSequence;
END_VAR

METHOD PUBLIC  GetAngle : LREAL
VAR_INPUT
	I : UINT;
END_VAR
VAR
	Angles : ARRAY [0..2] OF LREAL;
END_VAR
IF I >= Length THEN
	GetAngle := 0;
	RETURN;
END_IF

GetAngle := Angles[I];
END_METHOD

METHOD PUBLIC  GetDimension : Dimension
VAR_INPUT
	I : UINT;
END_VAR
VAR
	Dims : ARRAY [0..2] OF Dimension;
END_VAR
IF I >= Length THEN
	GetDimension := 0;
	RETURN;
END_IF

Dims := GetDimensions();
GetDimension := Dims[I];
END_METHOD

METHOD PUBLIC GetDimensions : ARRAY [0..2] OF Dimension
VAR_INPUT
END_VAR
CASE Sequence OF
	EulerAngleSequence.XYX:
		GetDimensions[0] := 0;
		GetDimensions[1] := 1;
		GetDimensions[2] := 0;
	EulerAngleSequence.XZX:
		GetDimensions[0] := 0;
		GetDimensions[1] := 2;
		GetDimensions[2] := 0;
	EulerAngleSequence.YXY:
		GetDimensions[0] := 1;
		GetDimensions[1] := 0;
		GetDimensions[2] := 1;
	EulerAngleSequence.YZY:
		GetDimensions[0] := 1;
		GetDimensions[1] := 2;
		GetDimensions[2] := 1;
	EulerAngleSequence.ZXZ:
		GetDimensions[0] := 2;
		GetDimensions[1] := 0;
		GetDimensions[2] := 2;
	EulerAngleSequence.ZYZ:
		GetDimensions[0] := 2;
		GetDimensions[1] := 1;
		GetDimensions[2] := 2;
	ELSE
		GetDimensions[0] := 0;
		GetDimensions[1] := 0;
		GetDimensions[2] := 0;
END_CASE
END_METHOD

PROPERTY Length : UINT
GET
Length := 3;
END_GET
END_PROPERTY

PROPERTY PUBLIC RaDeg : LREAL
GET
RaDeg := 180 * Angles_[0] / PI;
END_GET
SET
Angles_[0] := PI * RaDeg / 180;
END_SET
END_PROPERTY

PROPERTY PUBLIC RaRad : LREAL
GET
RaRad := Angles_[0];
END_GET
SET
Angles_[0] := RaRad;
END_SET
END_PROPERTY

PROPERTY PUBLIC RbDeg : LREAL
GET
RbDeg := 180 * Angles_[1] / PI;
END_GET
SET
Angles_[1] := PI * RbDeg / 180;
END_SET
END_PROPERTY

PROPERTY PUBLIC RbRad : LREAL
GET
RbRad := Angles_[1];
END_GET
SET
Angles_[1] := RbRad;
END_SET
END_PROPERTY

PROPERTY PUBLIC RcDeg : LREAL
GET
RcDeg := 180 * Angles_[2] / PI;
END_GET
SET
Angles_[2] := PI * RcDeg / 180;
END_SET
END_PROPERTY

PROPERTY PUBLIC RcRad : LREAL
GET
RcRad := Angles_[2];
END_GET
SET
Angles_[2] := RcRad;
END_SET
END_PROPERTY

PROPERTY PUBLIC Sequence : EulerAngleSequence
GET
Sequence := Sequence_;
END_GET
SET
Sequence_ := Sequence;
END_SET
END_PROPERTY

METHOD PUBLIC Clear
VAR_INPUT
END_VAR
Angles_[0] := 0;
Angles_[1] := 0;
Angles_[2] := 0;
END_METHOD

METHOD PUBLIC CopyFrom
VAR_INPUT
	O : EulerAngleOrientation;
END_VAR
CLEAR();
Sequence := O.Sequence;
AngleAccessor.CopyFrom(O.AngleAccessor);
END_METHOD

METHOD PUBLIC  SetAngle : BOOL
VAR_INPUT
	I : UINT;
	Val : LREAL;
END_VAR
VAR
	Angles : ARRAY [0..2] OF LREAL;
END_VAR
IF I >= Length THEN
	GetAngle := 0;
	SetAngle := FALSE;
	RETURN;
END_IF

SetAngle := TRUE;
Angles_[I] := Val;
END_METHOD

METHOD PUBLIC SetFromComponentsDeg
VAR_INPUT
	Ra : LREAL;
	Rb : LREAL;
	Rc : LREAL;
	Seq : EulerAngleSequence;
END_VAR
RaDeg := Ra;
RbDeg := Rb;
RcDeg := Rc;
Sequence := Seq;
END_METHOD

METHOD PUBLIC SetFromComponentsRad
VAR_INPUT
	Ra : LREAL;
	Rb : LREAL;
	Rc : LREAL;
	Seq : EulerAngleSequence;
END_VAR
RaRad := Ra;
RbRad := Rb;
RcRad := Rc;
Sequence := Seq;
END_METHOD

END_FUNCTION_BLOCK

// POUs/AngleSequence/IAngleSequenceOrientation
INTERFACE IAngleSequenceOrientation

END_INTERFACE
